// TIA Portal V18 export
// export: Created 2025-12-01T12:38:52.0419064Z, ExportSetting None, DisplayName Totally Integrated Automation Portal, DisplayVersion V18 Update 5, DisplayName TIA Portal Openness, DisplayVersion V18 Update 5, DisplayName TIA Portal Teamcenter Gateway, DisplayVersion V18, DisplayName TIA Portal Version Control Interface, DisplayVersion V18, DisplayName STEP 7 Professional, DisplayVersion V18 Update 5, DisplayName STEP 7 Safety, DisplayVersion V18, DisplayName WinCC Professional, DisplayVersion V18 Update 5
FUNCTION "MES" : Void   // FC500, LAD
{ S7_Optimized_Access := 'TRUE' }
// stored: AutoNumber false, SetENOAutomatically false
   VAR_TEMP
      YEAR : Int;
      MONTH : Int;
      DAY : Int;
      HH : Int;
      MM : Int;
      SS : Int;
      RET1 : Int;
      RET2 : Int;
      P : Array[0..10] of Bool;
   END_VAR
   VAR_TEMP   // added for the SCL form of the ladder/FBD networks
      _w1 : Bool;
      _w2 : Bool;
   END_VAR
BEGIN

REGION Network 2: 自动复位测试 / Automatic reset test
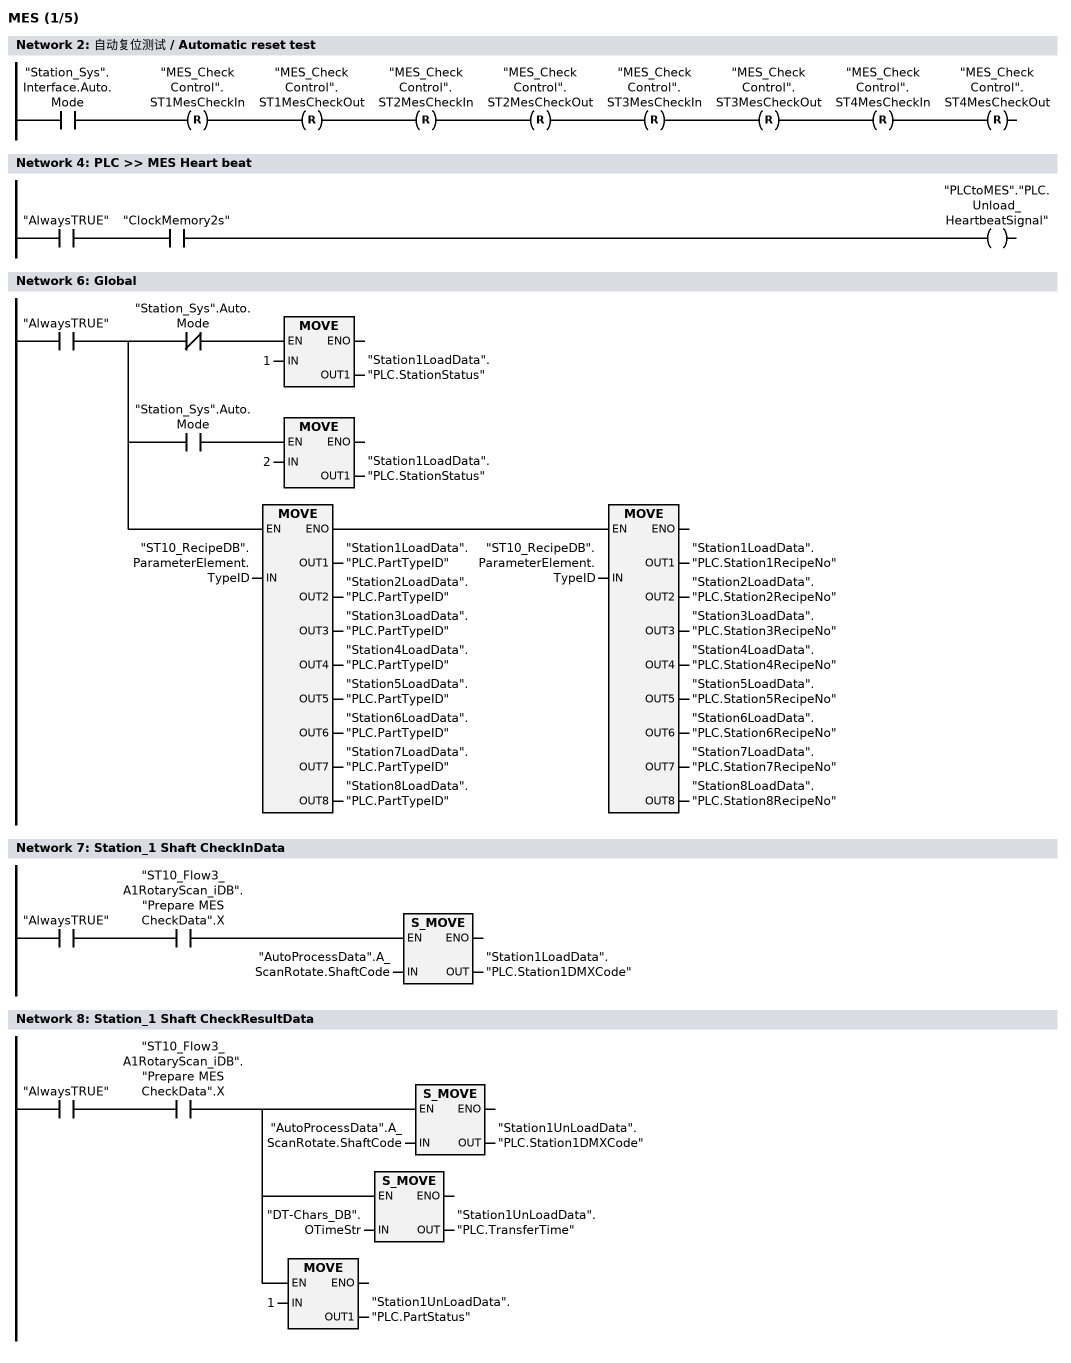
   RUNG wire#powerrail
      Contact( "Station_Sys".Interface.Auto.Mode )
      R_Coil( "MES_CheckControl".ST1MesCheckIn )
      R_Coil( "MES_CheckControl".ST1MesCheckOut )
      R_Coil( "MES_CheckControl".ST2MesCheckIn )
      R_Coil( "MES_CheckControl".ST2MesCheckOut )
      R_Coil( "MES_CheckControl".ST3MesCheckIn )
      R_Coil( "MES_CheckControl".ST3MesCheckOut )
      R_Coil( "MES_CheckControl".ST4MesCheckIn )
      R_Coil( "MES_CheckControl".ST4MesCheckOut )
   END_RUNG
   // the same network as SCL:
   IF "Station_Sys".Interface.Auto.Mode THEN
       "MES_CheckControl".ST1MesCheckIn := FALSE;
       "MES_CheckControl".ST1MesCheckOut := FALSE;
       "MES_CheckControl".ST2MesCheckIn := FALSE;
       "MES_CheckControl".ST2MesCheckOut := FALSE;
       "MES_CheckControl".ST3MesCheckIn := FALSE;
       "MES_CheckControl".ST3MesCheckOut := FALSE;
       "MES_CheckControl".ST4MesCheckIn := FALSE;
       "MES_CheckControl".ST4MesCheckOut := FALSE;
   END_IF;
END_REGION

NETWORK
TITLE = PLC系统时间转换 / PLC system time conversion
//########提取PLC当前日期
      L     %DB3000.DBB18;
      BTI;
      T     #YEAR;
      L     %DB3000.DBB19;
      BTI;
      T     #MONTH;
      L     %DB3000.DBB20;
      BTI;
      T     #DAY;
      L     %DB3000.DBB21;
      BTI;
      T     #HH;
      L     %DB3000.DBB22;
      BTI;
      T     #MM;
      L     %DB3000.DBB23;
      BTI;
      T     #SS;


//########将日期转化成字符
      CALL  "DT-Chars", "DT-Chars_DB"
      ( YEAR                := #YEAR,
        MONTH               := #MONTH,
        DAY                 := #DAY,
        HH                  := #HH,
        MM                  := #MM,
        SS                  := #SS,
        Year_Byte1          := ,
        Year_Byte2          := ,
        Month_Byte1         := ,
        Month_Byte2         := ,
        Days_Byte1          := ,
        Days_Byte2          := ,
        HH_Byte1            := ,
        HH_Byte2            := ,
        MM_Byte1            := ,
        MM_Byte2            := ,
        SS_Byte1            := ,
        SS_Byte2            := ,
        CalculateDays_Byte1 := ,
        CalculateDays_Byte2 := ,
        CalculateDays_Byte3 := ,
        Error_Code          := ,
        Year_Byte3          := ,
        Year_Byte4          := ,
        Month_Byte3         := ,
        Month_Byte4         := ,
        Days_Byte3          := ,
        Days_Byte4          := ,
        HH_Byte3            := ,
        HH_Byte4            := ,
        MM_Byte3            := ,
        MM_Byte4            := ,
        SS_Byte3            := ,
        SS_Byte4            := ,
        CalculateDays_Byte4 := ,
        CalculateDays_Byte5 := ,
        CalculateDays_Byte6 := ,
        OTimeStr            := 
      );




REGION Network 4: PLC >> MES Heart beat
   RUNG wire#powerrail
      Contact( "AlwaysTRUE" )
      Contact( "ClockMemory2s" )
      Coil( "PLCtoMES"."PLC.Unload_HeartbeatSignal" )
   END_RUNG
   // the same network as SCL:
   "PLCtoMES"."PLC.Unload_HeartbeatSignal" := "AlwaysTRUE" AND "ClockMemory2s";
END_REGION

REGION Network 6: Global
   RUNG wire#powerrail
      Contact( "AlwaysTRUE" )
      wire#w1
      I_Contact( "Station_Sys".Auto.Mode )
      Move(in := 1, out1 => "Station1LoadData"."PLC.StationStatus")
   END_RUNG
   RUNG wire#w1
      Contact( "Station_Sys".Auto.Mode )
      Move(in := 2, out1 => "Station1LoadData"."PLC.StationStatus")
   END_RUNG
   RUNG wire#w1
      Move(in := "ST10_RecipeDB".ParameterElement.TypeID, out1 => "Station1LoadData"."PLC.PartTypeID", out2 => "Station2LoadData"."PLC.PartTypeID", out3 => "Station3LoadData"."PLC.PartTypeID", out4 => "Station4LoadData"."PLC.PartTypeID", out5 => "Station5LoadData"."PLC.PartTypeID", out6 => "Station6LoadData"."PLC.PartTypeID", out7 => "Station7LoadData"."PLC.PartTypeID", out8 => "Station8LoadData"."PLC.PartTypeID")
      Move(in := "ST10_RecipeDB".ParameterElement.TypeID, out1 => "Station1LoadData"."PLC.Station1RecipeNo", out2 => "Station2LoadData"."PLC.Station2RecipeNo", out3 => "Station3LoadData"."PLC.Station3RecipeNo", out4 => "Station4LoadData"."PLC.Station4RecipeNo", out5 => "Station5LoadData"."PLC.Station5RecipeNo", out6 => "Station6LoadData"."PLC.Station6RecipeNo", out7 => "Station7LoadData"."PLC.Station7RecipeNo", out8 => "Station8LoadData"."PLC.Station8RecipeNo")
   END_RUNG
   // the same network as SCL:
   IF "AlwaysTRUE" AND NOT "Station_Sys".Auto.Mode THEN "Station1LoadData"."PLC.StationStatus" := 1; END_IF;
   IF "AlwaysTRUE" AND "Station_Sys".Auto.Mode THEN "Station1LoadData"."PLC.StationStatus" := 2; END_IF;
   IF "AlwaysTRUE" THEN
       "Station1LoadData"."PLC.PartTypeID" := "ST10_RecipeDB".ParameterElement.TypeID;
       "Station2LoadData"."PLC.PartTypeID" := "ST10_RecipeDB".ParameterElement.TypeID;
       "Station3LoadData"."PLC.PartTypeID" := "ST10_RecipeDB".ParameterElement.TypeID;
       "Station4LoadData"."PLC.PartTypeID" := "ST10_RecipeDB".ParameterElement.TypeID;
       "Station5LoadData"."PLC.PartTypeID" := "ST10_RecipeDB".ParameterElement.TypeID;
       "Station6LoadData"."PLC.PartTypeID" := "ST10_RecipeDB".ParameterElement.TypeID;
       "Station7LoadData"."PLC.PartTypeID" := "ST10_RecipeDB".ParameterElement.TypeID;
       "Station8LoadData"."PLC.PartTypeID" := "ST10_RecipeDB".ParameterElement.TypeID;
       "Station1LoadData"."PLC.Station1RecipeNo" := "ST10_RecipeDB".ParameterElement.TypeID;
       "Station2LoadData"."PLC.Station2RecipeNo" := "ST10_RecipeDB".ParameterElement.TypeID;
       "Station3LoadData"."PLC.Station3RecipeNo" := "ST10_RecipeDB".ParameterElement.TypeID;
       "Station4LoadData"."PLC.Station4RecipeNo" := "ST10_RecipeDB".ParameterElement.TypeID;
       "Station5LoadData"."PLC.Station5RecipeNo" := "ST10_RecipeDB".ParameterElement.TypeID;
       "Station6LoadData"."PLC.Station6RecipeNo" := "ST10_RecipeDB".ParameterElement.TypeID;
       "Station7LoadData"."PLC.Station7RecipeNo" := "ST10_RecipeDB".ParameterElement.TypeID;
       "Station8LoadData"."PLC.Station8RecipeNo" := "ST10_RecipeDB".ParameterElement.TypeID;
   END_IF;
END_REGION

REGION Network 7: Station_1 Shaft CheckInData
   RUNG wire#powerrail
      Contact( "AlwaysTRUE" )
      Contact( "ST10_Flow3_A1RotaryScan_iDB"."Prepare MES CheckData".X )
      S_Move(in := "AutoProcessData".A_ScanRotate.ShaftCode, out => "Station1LoadData"."PLC.Station1DMXCode")
   END_RUNG
   // the same network as SCL:
   IF "AlwaysTRUE" AND "ST10_Flow3_A1RotaryScan_iDB"."Prepare MES CheckData".X THEN
       "Station1LoadData"."PLC.Station1DMXCode" := "AutoProcessData".A_ScanRotate.ShaftCode;
   END_IF;
END_REGION

REGION Network 8: Station_1 Shaft CheckResultData
   RUNG wire#powerrail
      Contact( "AlwaysTRUE" )
      Contact( "ST10_Flow3_A1RotaryScan_iDB"."Prepare MES CheckData".X )
      wire#w1
      S_Move(in := "AutoProcessData".A_ScanRotate.ShaftCode, out => "Station1UnLoadData"."PLC.Station1DMXCode")
   END_RUNG
   RUNG wire#w1
      S_Move(in := "DT-Chars_DB".OTimeStr, out => "Station1UnLoadData"."PLC.TransferTime")
   END_RUNG
   RUNG wire#w1
      Move(in := 1, out1 => "Station1UnLoadData"."PLC.PartStatus")
   END_RUNG
   // the same network as SCL:
   IF "AlwaysTRUE" AND "ST10_Flow3_A1RotaryScan_iDB"."Prepare MES CheckData".X THEN
       "Station1UnLoadData"."PLC.Station1DMXCode" := "AutoProcessData".A_ScanRotate.ShaftCode;
       "Station1UnLoadData"."PLC.TransferTime" := "DT-Chars_DB".OTimeStr;
       "Station1UnLoadData"."PLC.PartStatus" := 1;
   END_IF;
END_REGION

REGION Network 10: Station_2 Ring_1 CheckInData
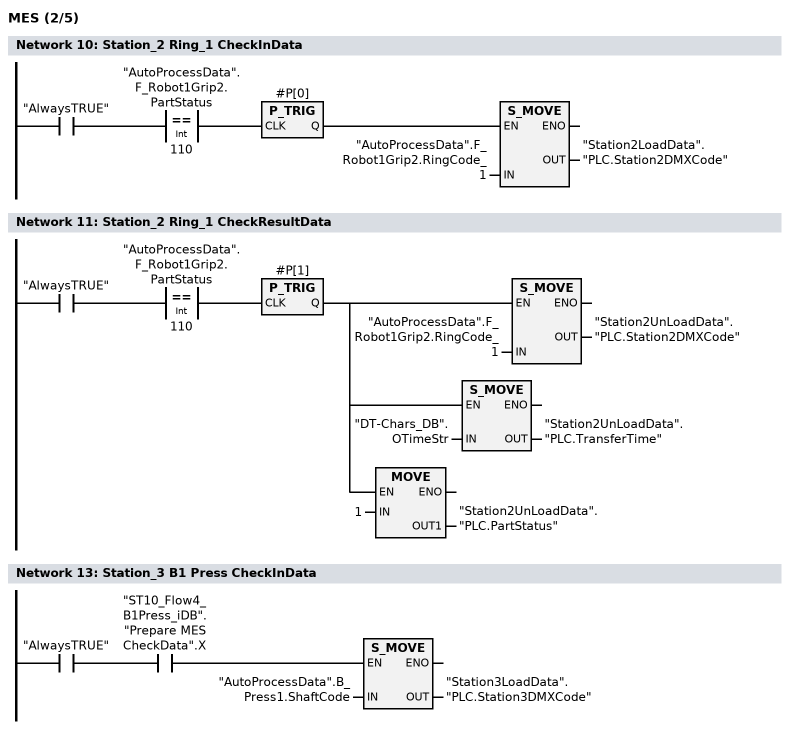
   RUNG wire#powerrail
      Contact( "AlwaysTRUE" )
      { S7_Templates := "SrcType := Int" } EQ_Contact(in1 := "AutoProcessData".F_Robot1Grip2.PartStatus, in2 := 110)
      P_Trig( #P[0] )
      S_Move(in := "AutoProcessData".F_Robot1Grip2.RingCode_1, out => "Station2LoadData"."PLC.Station2DMXCode")
   END_RUNG
   // the same network as SCL:
   #_w1 := "AlwaysTRUE" AND ("AutoProcessData".F_Robot1Grip2.PartStatus = 110);
   #_w2 := #_w1 AND NOT #P[0];   // rising edge
   #P[0] := #_w1;
   IF #_w2 THEN
       "Station2LoadData"."PLC.Station2DMXCode" := "AutoProcessData".F_Robot1Grip2.RingCode_1;
   END_IF;
END_REGION

REGION Network 11: Station_2 Ring_1 CheckResultData
   RUNG wire#powerrail
      Contact( "AlwaysTRUE" )
      { S7_Templates := "SrcType := Int" } EQ_Contact(in1 := "AutoProcessData".F_Robot1Grip2.PartStatus, in2 := 110)
      P_Trig( #P[1] )
      wire#w1
      S_Move(in := "AutoProcessData".F_Robot1Grip2.RingCode_1, out => "Station2UnLoadData"."PLC.Station2DMXCode")
   END_RUNG
   RUNG wire#w1
      S_Move(in := "DT-Chars_DB".OTimeStr, out => "Station2UnLoadData"."PLC.TransferTime")
   END_RUNG
   RUNG wire#w1
      Move(in := 1, out1 => "Station2UnLoadData"."PLC.PartStatus")
   END_RUNG
   // the same network as SCL:
   #_w1 := "AlwaysTRUE" AND ("AutoProcessData".F_Robot1Grip2.PartStatus = 110);
   #_w2 := #_w1 AND NOT #P[1];   // rising edge
   #P[1] := #_w1;
   IF #_w2 THEN
       "Station2UnLoadData"."PLC.Station2DMXCode" := "AutoProcessData".F_Robot1Grip2.RingCode_1;
       "Station2UnLoadData"."PLC.TransferTime" := "DT-Chars_DB".OTimeStr;
       "Station2UnLoadData"."PLC.PartStatus" := 1;
   END_IF;
END_REGION

REGION Network 13: Station_3 B1 Press CheckInData
   RUNG wire#powerrail
      Contact( "AlwaysTRUE" )
      Contact( "ST10_Flow4_B1Press_iDB"."Prepare MES CheckData".X )
      S_Move(in := "AutoProcessData".B_Press1.ShaftCode, out => "Station3LoadData"."PLC.Station3DMXCode")
   END_RUNG
   // the same network as SCL:
   IF "AlwaysTRUE" AND "ST10_Flow4_B1Press_iDB"."Prepare MES CheckData".X THEN
       "Station3LoadData"."PLC.Station3DMXCode" := "AutoProcessData".B_Press1.ShaftCode;
   END_IF;
END_REGION

REGION Network 14: Station_3 B1 Press CheckResultData
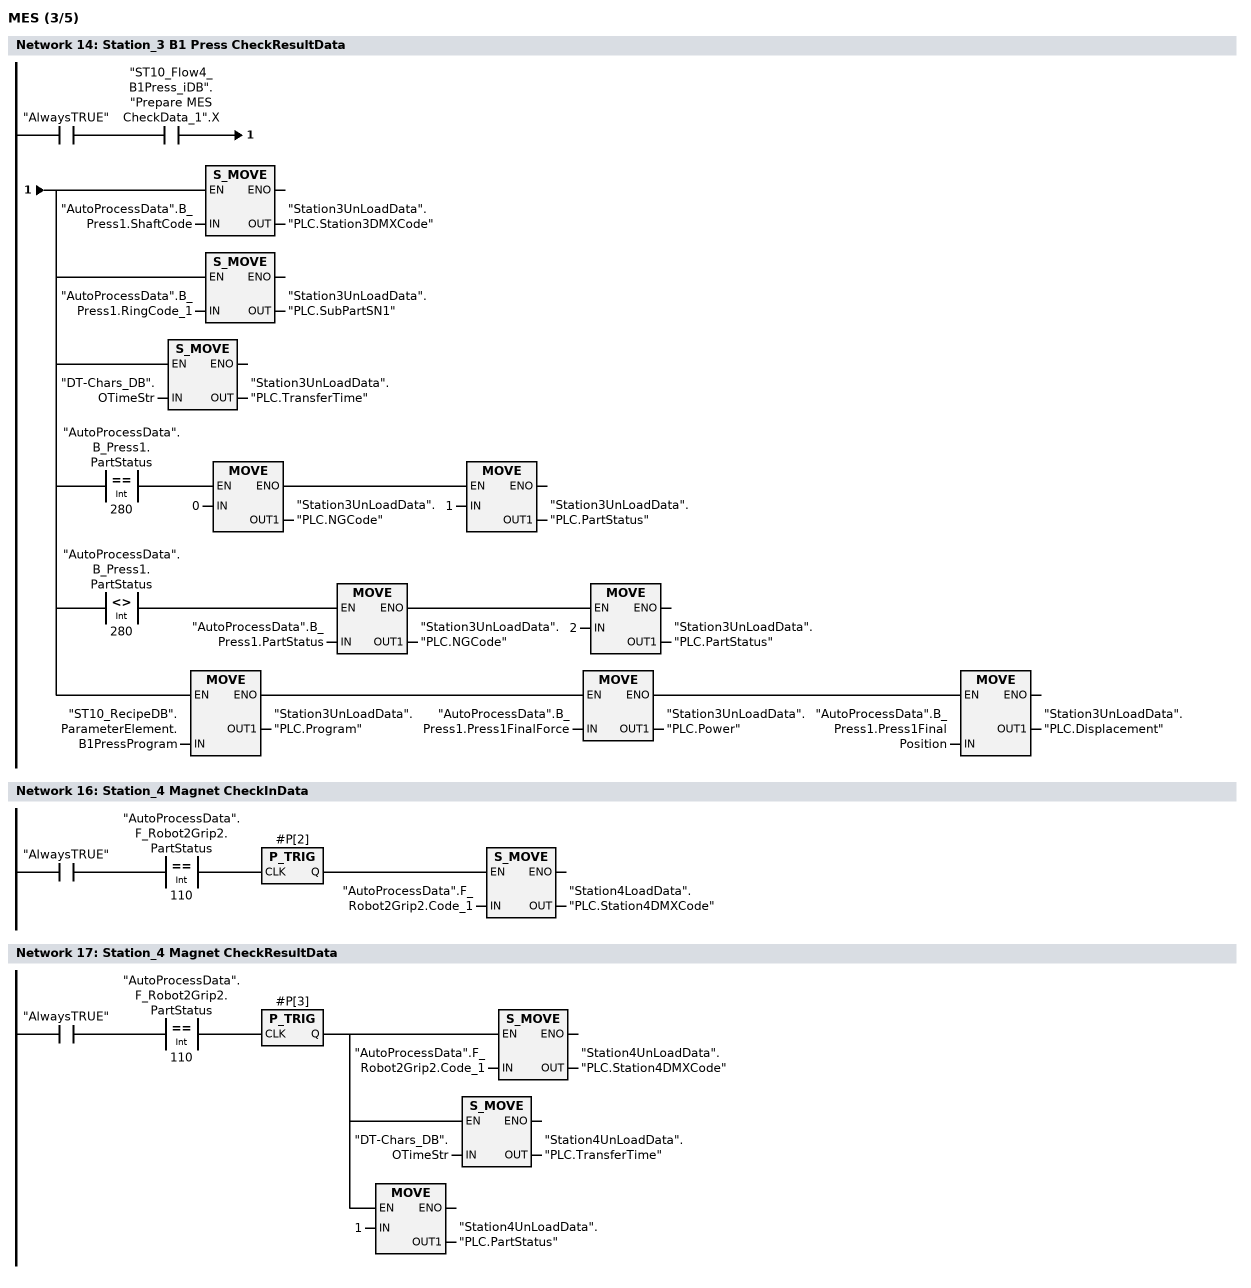
   RUNG wire#powerrail
      Contact( "AlwaysTRUE" )
      Contact( "ST10_Flow4_B1Press_iDB"."Prepare MES CheckData_1".X )
      wire#w1
      S_Move(in := "AutoProcessData".B_Press1.ShaftCode, out => "Station3UnLoadData"."PLC.Station3DMXCode")
   END_RUNG
   RUNG wire#w1
      S_Move(in := "AutoProcessData".B_Press1.RingCode_1, out => "Station3UnLoadData"."PLC.SubPartSN1")
   END_RUNG
   RUNG wire#w1
      S_Move(in := "DT-Chars_DB".OTimeStr, out => "Station3UnLoadData"."PLC.TransferTime")
   END_RUNG
   RUNG wire#w1
      { S7_Templates := "SrcType := Int" } EQ_Contact(in1 := "AutoProcessData".B_Press1.PartStatus, in2 := 280)
      Move(in := 0, out1 => "Station3UnLoadData"."PLC.NGCode")
      Move(in := 1, out1 => "Station3UnLoadData"."PLC.PartStatus")
   END_RUNG
   RUNG wire#w1
      { S7_Templates := "SrcType := Int" } NE_Contact(in1 := "AutoProcessData".B_Press1.PartStatus, in2 := 280)
      Move(in := "AutoProcessData".B_Press1.PartStatus, out1 => "Station3UnLoadData"."PLC.NGCode")
      Move(in := 2, out1 => "Station3UnLoadData"."PLC.PartStatus")
   END_RUNG
   RUNG wire#w1
      Move(in := "ST10_RecipeDB".ParameterElement.B1PressProgram, out1 => "Station3UnLoadData"."PLC.Program")
      Move(in := "AutoProcessData".B_Press1.Press1FinalForce, out1 => "Station3UnLoadData"."PLC.Power")
      Move(in := "AutoProcessData".B_Press1.Press1FinalPosition, out1 => "Station3UnLoadData"."PLC.Displacement")
   END_RUNG
   // the same network as SCL:
   #_w1 := "AlwaysTRUE" AND "ST10_Flow4_B1Press_iDB"."Prepare MES CheckData_1".X;
   IF #_w1 THEN
       "Station3UnLoadData"."PLC.Station3DMXCode" := "AutoProcessData".B_Press1.ShaftCode;
       "Station3UnLoadData"."PLC.SubPartSN1" := "AutoProcessData".B_Press1.RingCode_1;
       "Station3UnLoadData"."PLC.TransferTime" := "DT-Chars_DB".OTimeStr;
   END_IF;
   IF #_w1 AND ("AutoProcessData".B_Press1.PartStatus = 280) THEN
       "Station3UnLoadData"."PLC.NGCode" := 0;
       "Station3UnLoadData"."PLC.PartStatus" := 1;
   END_IF;
   IF #_w1 AND ("AutoProcessData".B_Press1.PartStatus <> 280) THEN
       "Station3UnLoadData"."PLC.NGCode" := "AutoProcessData".B_Press1.PartStatus;
       "Station3UnLoadData"."PLC.PartStatus" := 2;
   END_IF;
   IF #_w1 THEN
       "Station3UnLoadData"."PLC.Program" := "ST10_RecipeDB".ParameterElement.B1PressProgram;
       "Station3UnLoadData"."PLC.Power" := "AutoProcessData".B_Press1.Press1FinalForce;
       "Station3UnLoadData"."PLC.Displacement" := "AutoProcessData".B_Press1.Press1FinalPosition;
   END_IF;
END_REGION

REGION Network 16: Station_4 Magnet CheckInData
   RUNG wire#powerrail
      Contact( "AlwaysTRUE" )
      { S7_Templates := "SrcType := Int" } EQ_Contact(in1 := "AutoProcessData".F_Robot2Grip2.PartStatus, in2 := 110)
      P_Trig( #P[2] )
      S_Move(in := "AutoProcessData".F_Robot2Grip2.Code_1, out => "Station4LoadData"."PLC.Station4DMXCode")
   END_RUNG
   // the same network as SCL:
   #_w1 := "AlwaysTRUE" AND ("AutoProcessData".F_Robot2Grip2.PartStatus = 110);
   #_w2 := #_w1 AND NOT #P[2];   // rising edge
   #P[2] := #_w1;
   IF #_w2 THEN "Station4LoadData"."PLC.Station4DMXCode" := "AutoProcessData".F_Robot2Grip2.Code_1; END_IF;
END_REGION

REGION Network 17: Station_4 Magnet CheckResultData
   RUNG wire#powerrail
      Contact( "AlwaysTRUE" )
      { S7_Templates := "SrcType := Int" } EQ_Contact(in1 := "AutoProcessData".F_Robot2Grip2.PartStatus, in2 := 110)
      P_Trig( #P[3] )
      wire#w1
      S_Move(in := "AutoProcessData".F_Robot2Grip2.Code_1, out => "Station4UnLoadData"."PLC.Station4DMXCode")
   END_RUNG
   RUNG wire#w1
      S_Move(in := "DT-Chars_DB".OTimeStr, out => "Station4UnLoadData"."PLC.TransferTime")
   END_RUNG
   RUNG wire#w1
      Move(in := 1, out1 => "Station4UnLoadData"."PLC.PartStatus")
   END_RUNG
   // the same network as SCL:
   #_w1 := "AlwaysTRUE" AND ("AutoProcessData".F_Robot2Grip2.PartStatus = 110);
   #_w2 := #_w1 AND NOT #P[3];   // rising edge
   #P[3] := #_w1;
   IF #_w2 THEN
       "Station4UnLoadData"."PLC.Station4DMXCode" := "AutoProcessData".F_Robot2Grip2.Code_1;
       "Station4UnLoadData"."PLC.TransferTime" := "DT-Chars_DB".OTimeStr;
       "Station4UnLoadData"."PLC.PartStatus" := 1;
   END_IF;
END_REGION

REGION Network 19: Station_5 Glue CheckInData
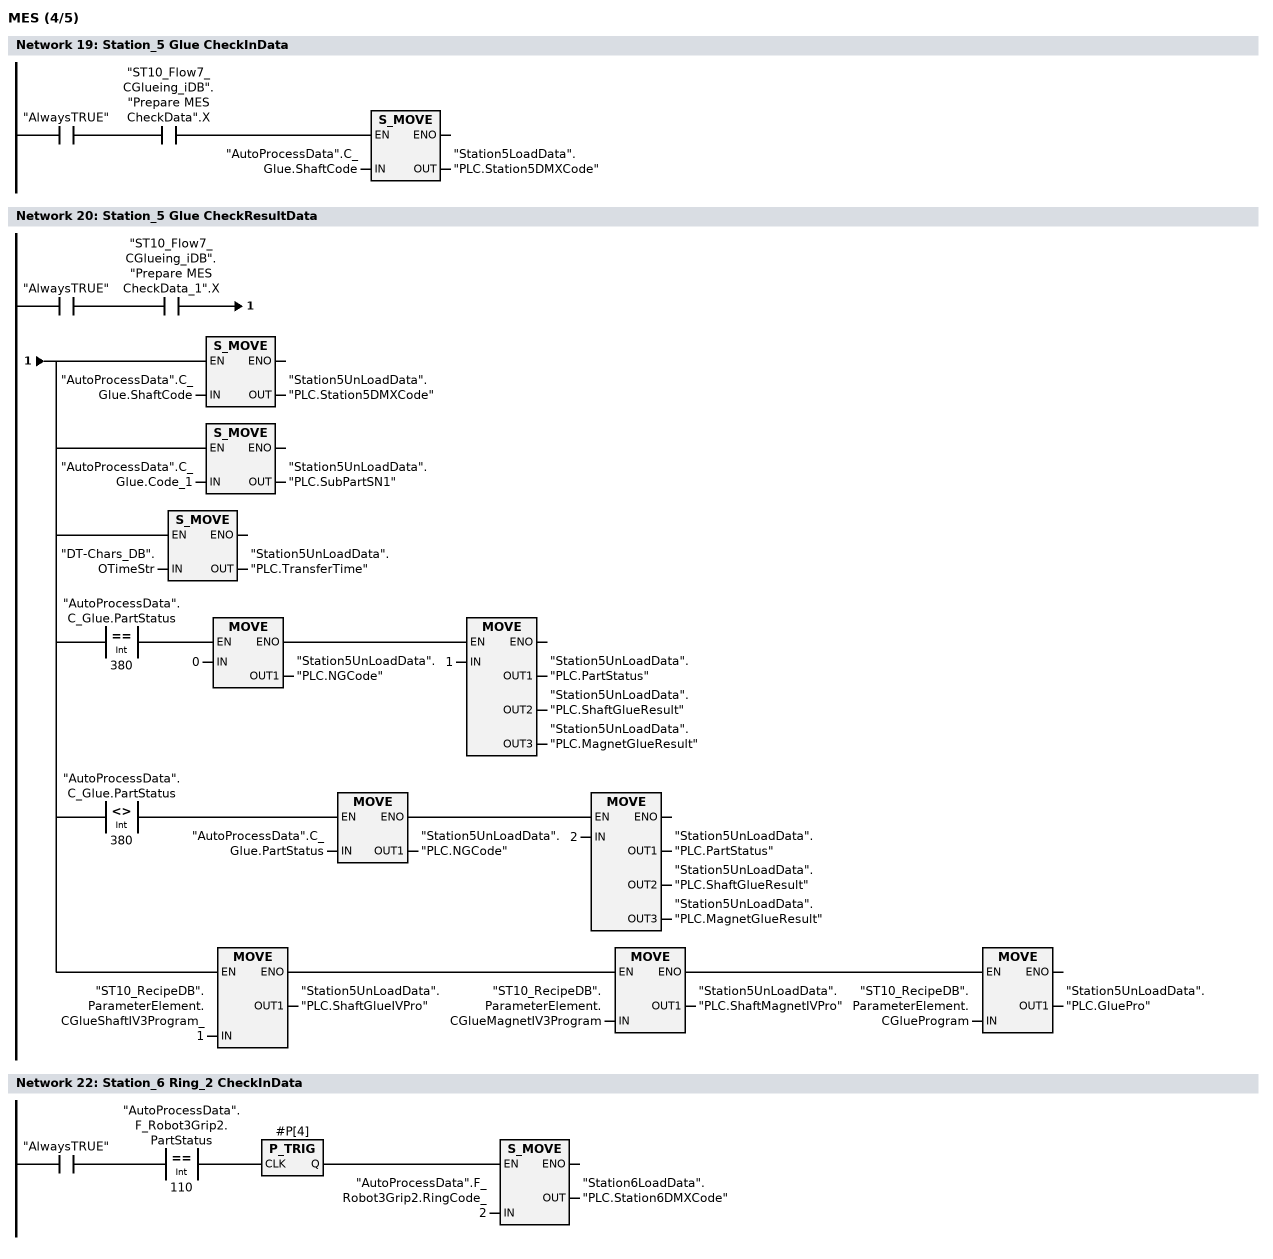
   RUNG wire#powerrail
      Contact( "AlwaysTRUE" )
      Contact( "ST10_Flow7_CGlueing_iDB"."Prepare MES CheckData".X )
      S_Move(in := "AutoProcessData".C_Glue.ShaftCode, out => "Station5LoadData"."PLC.Station5DMXCode")
   END_RUNG
   // the same network as SCL:
   IF "AlwaysTRUE" AND "ST10_Flow7_CGlueing_iDB"."Prepare MES CheckData".X THEN
       "Station5LoadData"."PLC.Station5DMXCode" := "AutoProcessData".C_Glue.ShaftCode;
   END_IF;
END_REGION

REGION Network 20: Station_5 Glue CheckResultData
   RUNG wire#powerrail
      Contact( "AlwaysTRUE" )
      Contact( "ST10_Flow7_CGlueing_iDB"."Prepare MES CheckData_1".X )
      wire#w1
      S_Move(in := "AutoProcessData".C_Glue.ShaftCode, out => "Station5UnLoadData"."PLC.Station5DMXCode")
   END_RUNG
   RUNG wire#w1
      S_Move(in := "AutoProcessData".C_Glue.Code_1, out => "Station5UnLoadData"."PLC.SubPartSN1")
   END_RUNG
   RUNG wire#w1
      S_Move(in := "DT-Chars_DB".OTimeStr, out => "Station5UnLoadData"."PLC.TransferTime")
   END_RUNG
   RUNG wire#w1
      { S7_Templates := "SrcType := Int" } EQ_Contact(in1 := "AutoProcessData".C_Glue.PartStatus, in2 := 380)
      Move(in := 0, out1 => "Station5UnLoadData"."PLC.NGCode")
      Move(in := 1, out1 => "Station5UnLoadData"."PLC.PartStatus", out2 => "Station5UnLoadData"."PLC.ShaftGlueResult", out3 => "Station5UnLoadData"."PLC.MagnetGlueResult")
   END_RUNG
   RUNG wire#w1
      { S7_Templates := "SrcType := Int" } NE_Contact(in1 := "AutoProcessData".C_Glue.PartStatus, in2 := 380)
      Move(in := "AutoProcessData".C_Glue.PartStatus, out1 => "Station5UnLoadData"."PLC.NGCode")
      Move(in := 2, out1 => "Station5UnLoadData"."PLC.PartStatus", out2 => "Station5UnLoadData"."PLC.ShaftGlueResult", out3 => "Station5UnLoadData"."PLC.MagnetGlueResult")
   END_RUNG
   RUNG wire#w1
      Move(in := "ST10_RecipeDB".ParameterElement.CGlueShaftIV3Program_1, out1 => "Station5UnLoadData"."PLC.ShaftGlueIVPro")
      Move(in := "ST10_RecipeDB".ParameterElement.CGlueMagnetIV3Program, out1 => "Station5UnLoadData"."PLC.ShaftMagnetIVPro")
      Move(in := "ST10_RecipeDB".ParameterElement.CGlueProgram, out1 => "Station5UnLoadData"."PLC.GluePro")
   END_RUNG
   // the same network as SCL:
   #_w1 := "AlwaysTRUE" AND "ST10_Flow7_CGlueing_iDB"."Prepare MES CheckData_1".X;
   IF #_w1 THEN
       "Station5UnLoadData"."PLC.Station5DMXCode" := "AutoProcessData".C_Glue.ShaftCode;
       "Station5UnLoadData"."PLC.SubPartSN1" := "AutoProcessData".C_Glue.Code_1;
       "Station5UnLoadData"."PLC.TransferTime" := "DT-Chars_DB".OTimeStr;
   END_IF;
   IF #_w1 AND ("AutoProcessData".C_Glue.PartStatus = 380) THEN
       "Station5UnLoadData"."PLC.NGCode" := 0;
       "Station5UnLoadData"."PLC.PartStatus" := 1;
       "Station5UnLoadData"."PLC.ShaftGlueResult" := 1;
       "Station5UnLoadData"."PLC.MagnetGlueResult" := 1;
   END_IF;
   IF #_w1 AND ("AutoProcessData".C_Glue.PartStatus <> 380) THEN
       "Station5UnLoadData"."PLC.NGCode" := "AutoProcessData".C_Glue.PartStatus;
       "Station5UnLoadData"."PLC.PartStatus" := 2;
       "Station5UnLoadData"."PLC.ShaftGlueResult" := 2;
       "Station5UnLoadData"."PLC.MagnetGlueResult" := 2;
   END_IF;
   IF #_w1 THEN
       "Station5UnLoadData"."PLC.ShaftGlueIVPro" := "ST10_RecipeDB".ParameterElement.CGlueShaftIV3Program_1;
       "Station5UnLoadData"."PLC.ShaftMagnetIVPro" := "ST10_RecipeDB".ParameterElement.CGlueMagnetIV3Program;
       "Station5UnLoadData"."PLC.GluePro" := "ST10_RecipeDB".ParameterElement.CGlueProgram;
   END_IF;
END_REGION

REGION Network 22: Station_6 Ring_2 CheckInData
   RUNG wire#powerrail
      Contact( "AlwaysTRUE" )
      { S7_Templates := "SrcType := Int" } EQ_Contact(in1 := "AutoProcessData".F_Robot3Grip2.PartStatus, in2 := 110)
      P_Trig( #P[4] )
      S_Move(in := "AutoProcessData".F_Robot3Grip2.RingCode_2, out => "Station6LoadData"."PLC.Station6DMXCode")
   END_RUNG
   // the same network as SCL:
   #_w1 := "AlwaysTRUE" AND ("AutoProcessData".F_Robot3Grip2.PartStatus = 110);
   #_w2 := #_w1 AND NOT #P[4];   // rising edge
   #P[4] := #_w1;
   IF #_w2 THEN
       "Station6LoadData"."PLC.Station6DMXCode" := "AutoProcessData".F_Robot3Grip2.RingCode_2;
   END_IF;
END_REGION

REGION Network 23: Station_6 Ring_2 CheckResultData
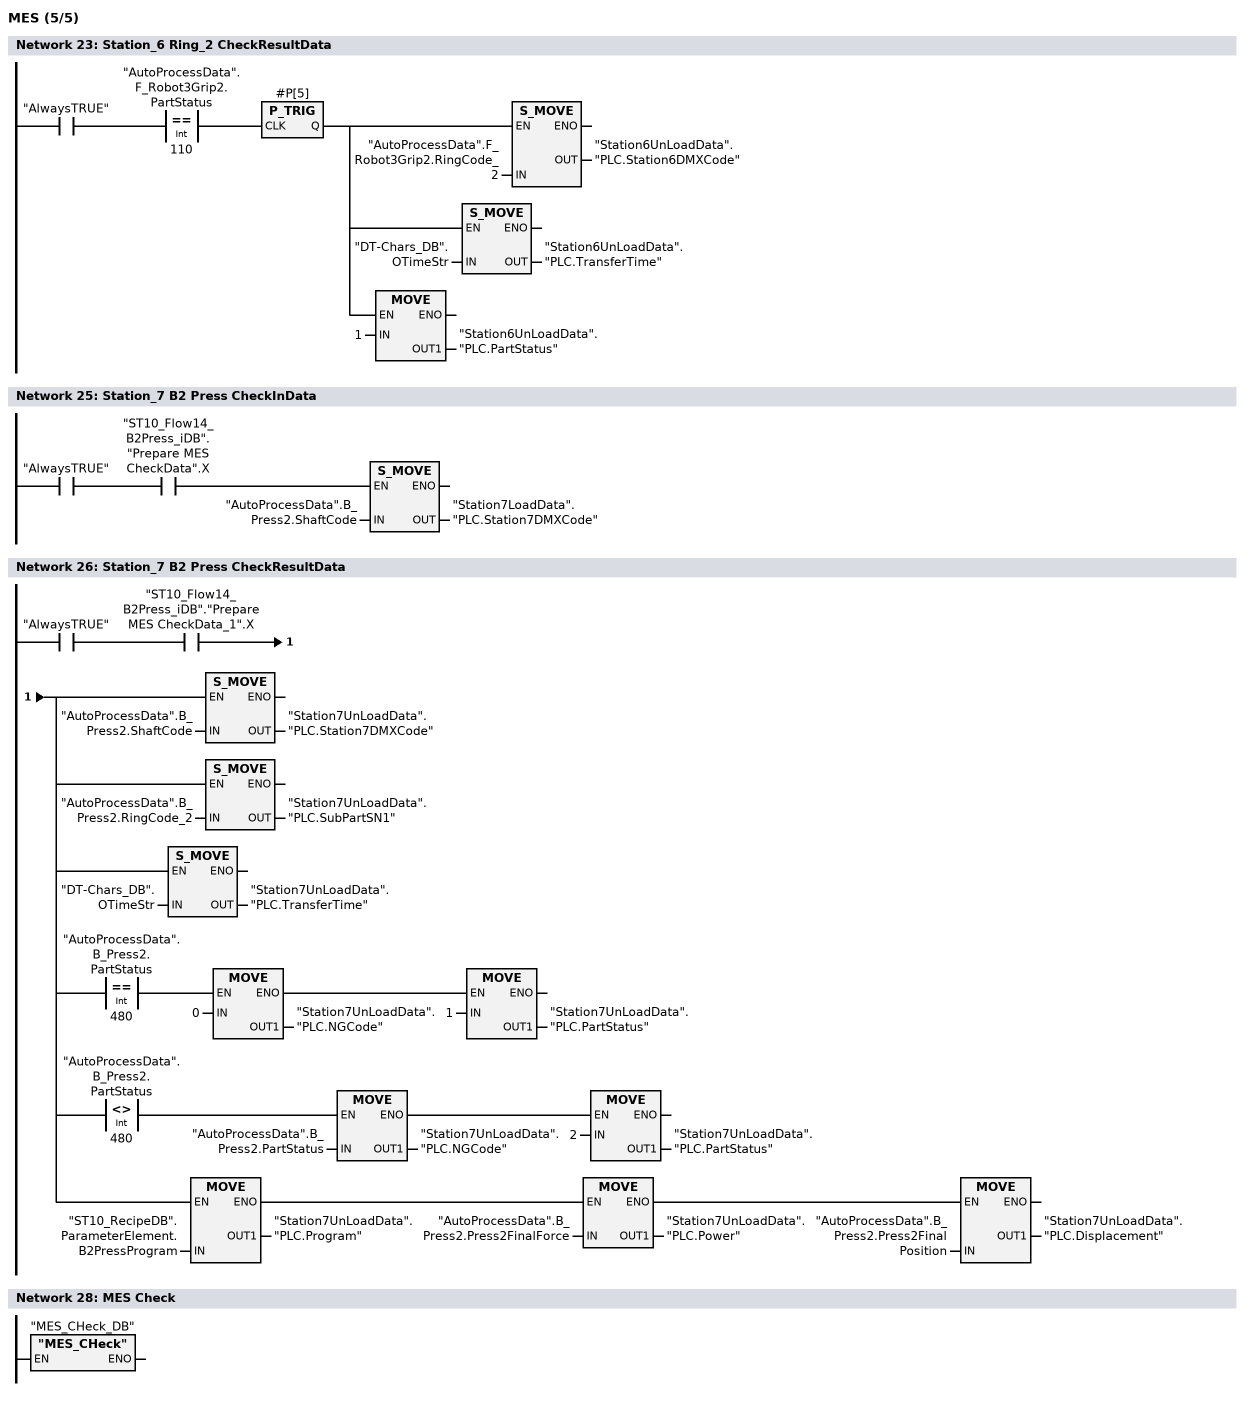
   RUNG wire#powerrail
      Contact( "AlwaysTRUE" )
      { S7_Templates := "SrcType := Int" } EQ_Contact(in1 := "AutoProcessData".F_Robot3Grip2.PartStatus, in2 := 110)
      P_Trig( #P[5] )
      wire#w1
      S_Move(in := "AutoProcessData".F_Robot3Grip2.RingCode_2, out => "Station6UnLoadData"."PLC.Station6DMXCode")
   END_RUNG
   RUNG wire#w1
      S_Move(in := "DT-Chars_DB".OTimeStr, out => "Station6UnLoadData"."PLC.TransferTime")
   END_RUNG
   RUNG wire#w1
      Move(in := 1, out1 => "Station6UnLoadData"."PLC.PartStatus")
   END_RUNG
   // the same network as SCL:
   #_w1 := "AlwaysTRUE" AND ("AutoProcessData".F_Robot3Grip2.PartStatus = 110);
   #_w2 := #_w1 AND NOT #P[5];   // rising edge
   #P[5] := #_w1;
   IF #_w2 THEN
       "Station6UnLoadData"."PLC.Station6DMXCode" := "AutoProcessData".F_Robot3Grip2.RingCode_2;
       "Station6UnLoadData"."PLC.TransferTime" := "DT-Chars_DB".OTimeStr;
       "Station6UnLoadData"."PLC.PartStatus" := 1;
   END_IF;
END_REGION

REGION Network 25: Station_7 B2 Press CheckInData
   RUNG wire#powerrail
      Contact( "AlwaysTRUE" )
      Contact( "ST10_Flow14_B2Press_iDB"."Prepare MES CheckData".X )
      S_Move(in := "AutoProcessData".B_Press2.ShaftCode, out => "Station7LoadData"."PLC.Station7DMXCode")
   END_RUNG
   // the same network as SCL:
   IF "AlwaysTRUE" AND "ST10_Flow14_B2Press_iDB"."Prepare MES CheckData".X THEN
       "Station7LoadData"."PLC.Station7DMXCode" := "AutoProcessData".B_Press2.ShaftCode;
   END_IF;
END_REGION

REGION Network 26: Station_7 B2 Press CheckResultData
   RUNG wire#powerrail
      Contact( "AlwaysTRUE" )
      Contact( "ST10_Flow14_B2Press_iDB"."Prepare MES CheckData_1".X )
      wire#w1
      S_Move(in := "AutoProcessData".B_Press2.ShaftCode, out => "Station7UnLoadData"."PLC.Station7DMXCode")
   END_RUNG
   RUNG wire#w1
      S_Move(in := "AutoProcessData".B_Press2.RingCode_2, out => "Station7UnLoadData"."PLC.SubPartSN1")
   END_RUNG
   RUNG wire#w1
      S_Move(in := "DT-Chars_DB".OTimeStr, out => "Station7UnLoadData"."PLC.TransferTime")
   END_RUNG
   RUNG wire#w1
      { S7_Templates := "SrcType := Int" } EQ_Contact(in1 := "AutoProcessData".B_Press2.PartStatus, in2 := 480)
      Move(in := 0, out1 => "Station7UnLoadData"."PLC.NGCode")
      Move(in := 1, out1 => "Station7UnLoadData"."PLC.PartStatus")
   END_RUNG
   RUNG wire#w1
      { S7_Templates := "SrcType := Int" } NE_Contact(in1 := "AutoProcessData".B_Press2.PartStatus, in2 := 480)
      Move(in := "AutoProcessData".B_Press2.PartStatus, out1 => "Station7UnLoadData"."PLC.NGCode")
      Move(in := 2, out1 => "Station7UnLoadData"."PLC.PartStatus")
   END_RUNG
   RUNG wire#w1
      Move(in := "ST10_RecipeDB".ParameterElement.B2PressProgram, out1 => "Station7UnLoadData"."PLC.Program")
      Move(in := "AutoProcessData".B_Press2.Press2FinalForce, out1 => "Station7UnLoadData"."PLC.Power")
      Move(in := "AutoProcessData".B_Press2.Press2FinalPosition, out1 => "Station7UnLoadData"."PLC.Displacement")
   END_RUNG
   // the same network as SCL:
   #_w1 := "AlwaysTRUE" AND "ST10_Flow14_B2Press_iDB"."Prepare MES CheckData_1".X;
   IF #_w1 THEN
       "Station7UnLoadData"."PLC.Station7DMXCode" := "AutoProcessData".B_Press2.ShaftCode;
       "Station7UnLoadData"."PLC.SubPartSN1" := "AutoProcessData".B_Press2.RingCode_2;
       "Station7UnLoadData"."PLC.TransferTime" := "DT-Chars_DB".OTimeStr;
   END_IF;
   IF #_w1 AND ("AutoProcessData".B_Press2.PartStatus = 480) THEN
       "Station7UnLoadData"."PLC.NGCode" := 0;
       "Station7UnLoadData"."PLC.PartStatus" := 1;
   END_IF;
   IF #_w1 AND ("AutoProcessData".B_Press2.PartStatus <> 480) THEN
       "Station7UnLoadData"."PLC.NGCode" := "AutoProcessData".B_Press2.PartStatus;
       "Station7UnLoadData"."PLC.PartStatus" := 2;
   END_IF;
   IF #_w1 THEN
       "Station7UnLoadData"."PLC.Program" := "ST10_RecipeDB".ParameterElement.B2PressProgram;
       "Station7UnLoadData"."PLC.Power" := "AutoProcessData".B_Press2.Press2FinalForce;
       "Station7UnLoadData"."PLC.Displacement" := "AutoProcessData".B_Press2.Press2FinalPosition;
   END_IF;
END_REGION

REGION Network 28: MES Check
   RUNG wire#powerrail
      "MES_CHeck_DB"()
   END_RUNG
   // the same network as SCL:
   "MES_CHeck_DB"();   // "MES_CHeck"
END_REGION
END_FUNCTION
